TYPE E_CommandStatus :
(
    CMDSTAT_IDLE        := 0,
    CMDSTAT_PENDING     := 1,
    CMDSTAT_EXECUTING   := 2,
    CMDSTAT_DONE        := 3,
    CMDSTAT_ERROR       := 4
);
END_TYPE

(* stored: Version 1.1.0.1
   DUT E_CommandStatus: Id {3BC6DE44-3108-AAC9-140D-E2E158E71B83} *)
